FUNCTION_BLOCK FB_HeightMeasurement
VAR_INPUT

	aSensorCurrentValue							: ARRAY[1..4] OF DINT;
	bEnable										: BOOL;
	bMeasurementRequest							: BOOL;
	
	
	bSet										: BOOL;
	aTolerance									: ARRAY[1..4] OF DINT;

	
	bManualMode									: BOOL;
	bManualMeasure								: BOOL;
	bAcknowledge								: BOOL;
	bFunctionFault								: BOOL;
	
	
	
	
END_VAR
VAR_OUTPUT
	bBusy										: BOOL;
	bComplete									: BOOL;
	bEnableo									: BOOL;
	wFunctionState								: STRING;
	nSensorSetPoint								: ARRAY[1..4] OF DINT;
	aPass										: ARRAY[1..5] OF BOOL; //5 Final Result
	aFail										: ARRAY[1..5] OF BOOL; //5 Final Result
	aMinLimit									: ARRAY[1..4] OF DINT;
	aMaxLimit									: ARRAY[1..4] OF DINT;

	
END_VAR
VAR
	i											: INT;
	j											: INT;
	nFunctionProcess							: INT;
	nReference									: DINT;
	
	tonCaseDelay								: ARRAY[0..10] OF TON;
	rtrigCaseTriger								: ARRAY[0..10] OF R_TRIG;
END_VAR

ACT_TimTrig();

IF NOT bEnable THEN
	nFunctionProcess			:= 0;
	bEnableo					:= FALSE;
ELSE 
	bEnableo					:= TRUE;
END_IF





CASE nFunctionProcess OF 

0:
wFunctionState				:='Function Disabled';
bBusy						:= FALSE;
IF bEnable THEN
	nFunctionProcess		:=1;
END_IF

1:
wFunctionState				:='Waiting';
IF tonCaseDelay[5].Q THEN
	nFunctionProcess		:=2;
END_IF
2:
j							:= 0;
ACT_Fault();
IF bFunctionFault THEN
	nFunctionProcess		:=50;
ELSIF bMeasurementRequest THEN
	nFunctionProcess		:=10;
ELSIF	bManualMode THEN
	nFunctionProcess		:=30;
END_IF

10:
j							:= 0;
FOR j:=1 TO 5 DO
	
	aPass[j] 				:= FALSE;
	aFail[j] 				:= FALSE;
	
END_FOR
IF tonCaseDelay[6].Q THEN
	nFunctionProcess		:=11;
END_IF
11:
wFunctionState				:='Working';
bBusy						:= TRUE;
IF tonCaseDelay[0].Q THEN
	nFunctionProcess		:=13;
END_IF

13:
FOR j:=1 TO 4 DO
	IF aSensorCurrentValue[j] < aMaxLimit[j] AND  aSensorCurrentValue[j] > aMinLimit[j] THEN
		aPass[j] := TRUE;
	ELSE aFail[j] := TRUE;
	END_IF
END_FOR
IF tonCaseDelay[1].Q THEN
	nFunctionProcess		:=14;
	j						:= 0;
END_IF

14:
aPass[5]					:= TRUE;
aFail[5]					:= FALSE;
FOR j:=1 TO 4 DO
IF aFail[j] THEN
	aPass[5]				:= FALSE;
	aFail[5]				:= TRUE;
END_IF
END_FOR
IF tonCaseDelay[3].Q THEN
	nFunctionProcess		:=16;
END_IF

16:
wFunctionState				:='Process Complete';
bComplete					:= TRUE;
bBusy						:= FALSE;
j							:= 0;
IF bAcknowledge  THEN	
	nFunctionProcess		:=20;
END_IF

20:
bComplete	:= FALSE;
IF tonCaseDelay[2].Q THEN
	nFunctionProcess		:=1;
END_IF

30:
wFunctionState				:='Manual Mode';
IF bManualMode THEN
	ACT_Manual();
ELSIF bFunctionFault THEN
	nFunctionProcess		:=50;
ELSE nFunctionProcess		:=1;
END_IF




50: 
wFunctionState				:='Error';
IF tonCaseDelay[4].Q THEN
	nFunctionProcess		:=1;
END_IF



END_CASE

ACTION ACT_Fault:
(*FOR i:=1 TO 5 DO
	IF aCurrentValueInvalid[i] OR aCurrentValueUnderRange[i] OR aCurrentValueOverRange[i] OR aSensorErrorStatus[i] OR bTerminalErrorStatus THEN 

	bFunctionFault := TRUE;
	
	ELSE bFunctionFault := FALSE;
	
	END_IF

END_FOR
IF GVL_MASTER.bFlash1Hz THEN
	i:=0;
END_IF*)
END_ACTION

ACTION ACT_Manual:
	

	aMinLimit[1]		:= nSensorSetPoint[1] - aTolerance[1];
	aMinLimit[2]		:= nSensorSetPoint[2] - aTolerance[2];
	aMinLimit[3]		:= nSensorSetPoint[3] - aTolerance[3];
	aMinLimit[4]		:= nSensorSetPoint[4] - aTolerance[4];
	
	aMaxLimit[1]		:= nSensorSetPoint[1] + aTolerance[1];
	aMaxLimit[2]		:= nSensorSetPoint[2] + aTolerance[2];
	aMaxLimit[3]		:= nSensorSetPoint[3] + aTolerance[3];
	aMaxLimit[4]		:= nSensorSetPoint[4] + aTolerance[4];

IF bSet THEN
	
	nSensorSetPoint[1] 	:= aSensorCurrentValue[1];
	nSensorSetPoint[2] 	:= aSensorCurrentValue[2];
	nSensorSetPoint[3] 	:= aSensorCurrentValue[3];
	nSensorSetPoint[4] 	:= aSensorCurrentValue[4];
	

	
END_IF

IF bManualMeasure THEN
	aPass[5]					:= TRUE;
	aFail[5]					:= FALSE;
	FOR j:=1 TO 4 DO
		IF aSensorCurrentValue[j] <= aMaxLimit[j] AND  aSensorCurrentValue[j] >= aMinLimit[j] THEN
			aPass[j] := TRUE;
			aFail[j] := FALSE;
		ELSE 
			aFail[j] := TRUE;
			aPass[j] := FALSE;
			
		END_IF
		IF aFail[j] THEN
		aPass[5]				:= FALSE;
		aFail[5]				:= TRUE;
		END_IF
	END_FOR
	

	
END_IF
END_ACTION

ACTION ACT_TimTrig:
tonCaseDelay[0](IN:= nFunctionProcess = 11,PT:=T#3S);
tonCaseDelay[1](IN:= nFunctionProcess = 13,PT:=T#1S);
tonCaseDelay[2](IN:= nFunctionProcess = 20,PT:=T#1S);
tonCaseDelay[3](IN:= nFunctionProcess = 14,PT:=T#1S);
tonCaseDelay[4](IN:= nFunctionProcess = 50 AND NOT bFunctionFault,PT:=T#1S);
tonCaseDelay[5](IN:= nFunctionProcess = 1,PT:=T#1S);
tonCaseDelay[6](IN:=nFunctionProcess = 10 ,PT:=T#1S);
tonCaseDelay[7](IN:= ,PT:=T#2S);

//rtrigCaseTriger[0]();
END_ACTION

END_FUNCTION_BLOCK

(* stored: Version 1.1.0.1, ProductVersion 3.1.4024.13
   POU FB_HeightMeasurement: Id {068aacf2-79ff-442c-ae13-d0bbf542e719}, SpecialFunc None
   Action ACT_Fault: Id {dd5f2a91-7d58-4671-82a8-3d6b14d909e6}
   Action ACT_Manual: Id {a603d0c8-21db-462b-b2f5-61c009f114aa}
   Action ACT_TimTrig: Id {6a19913a-a816-4bfe-a146-bb743b608325} *)
